{attribute 'GeneratedUsingTerminal: ELX3202-0000-0016'}
{attribute addProperty BoxType "ELX3202-0000-0016"}
{attribute addProperty Id "RTD_Inputs_Channel_1AT %I*RTD_Inputs_Channel_4A3944819RTD_Inputs_Channel_2AT %I*RTD_Inputs_Channel_4A3944819WcStateAT %I*WcState_9091E0EB2InfoDataAT %I*InfoData_32EB74EA10"}
{attribute addProperty CRC "682269165"}
{attribute addProperty Size "30"}
TYPE ELX3202_28AA99ED EXTENDS EtcSlaveTerminalBase_947E5A46 :
STRUCT
	{attribute addProperty Name "RTD_Inputs_Channel_1"}
	RTD_Inputs_Channel_1 : RTD_Inputs_Channel_4A394481;
	{attribute addProperty Name "RTD_Inputs_Channel_2"}
	RTD_Inputs_Channel_2 : RTD_Inputs_Channel_4A394481;
	{attribute addProperty Name "WcState"}
	WcState : WcState_9091E0EB;
	{attribute addProperty Name "InfoData"}
	InfoData : InfoData_32EB74EA;
END_STRUCT
END_TYPE

(* stored: Version 1.2.0.0, ProductVersion 3.1.4024.9
   DUT ELX3202_28AA99ED: Id {8ca89f02-079d-4bb3-a16c-9ca3ac3aefe5} *)
